TYPE ST_CoolingSystem_Inputs :
STRUCT
	BattLoopValveFB					:	BOOL;
	InvLoopValveFB					:	BOOL;
	FancoilLoopValveFB				:	BOOL;
	
	CoolingLoopPressureSensor 		:	INT;
	CoolingLoopTemperatureSensor 	:	INT;
	
	CoolingSystem400VFuseFB			:	BOOL;
	ACPumpFb						: 	BOOL;
	
END_STRUCT
END_TYPE

(* stored: Version 1.1.0.1, ProductVersion 3.1.4024.12
   DUT ST_CoolingSystem_Inputs: Id {0bb2d494-187a-443e-b7e4-c37368189fc9} *)
